(* PLC project mixture, Dassault Systèmes ControlBuild 2024x *)
(* stored: creationDateTime 2023-10-03T11:13:39-01:00 *)

FUNCTION_BLOCK faults
  VAR_INPUT
    generalFault1 : BOOL := false;
    generalFault2 : BOOL := false;
    generalFault3 : BOOL := false;
  END_VAR
  VAR_OUTPUT
    fault : BOOL := false;
  END_VAR

(* LD diagram, written out as Structured Text *)
1:
fault := generalFault3 OR generalFault1 OR generalFault2;
END_FUNCTION_BLOCK

PROGRAM batch.mixture
  VAR_INPUT
    cycleInProgress : BOOL := false;
    kneadingRequest : BOOL := false;
    acknowledgePB : BOOL := false;
  END_VAR
  VAR_INPUT
    autoMode : BOOL := false;
    manualMode : BOOL := false;
  END_VAR
  VAR_INPUT
    syrupExtraction : REAL := 0.0;
    flourExtraction : REAL := 0.0;
  END_VAR
  VAR_OUTPUT
    kneadingOK : BOOL := false;
    fault : BOOL := false;
  END_VAR

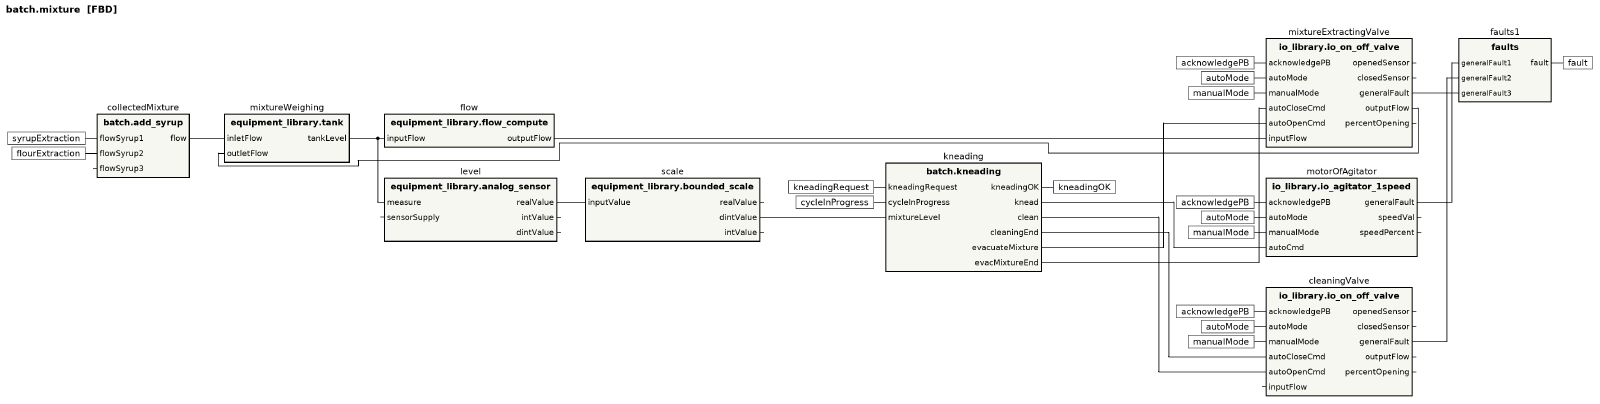
(* FBD diagram, written out as Structured Text *)
collectedMixture(flowSyrup1 := syrupExtraction, flowSyrup2 := flourExtraction);
flow(inputFlow := mixtureWeighing.tankLevel);
mixtureExtractingValve(acknowledgePB := acknowledgePB, autoMode := autoMode, manualMode := manualMode, autoCloseCmd := kneading.evacMixtureEnd, autoOpenCmd := kneading.evacuateMixture, inputFlow := flow.outputFlow);
mixtureWeighing(inletFlow := collectedMixture.flow, outletFlow := mixtureExtractingValve.outputFlow);
level(measure := mixtureWeighing.tankLevel);
scale(inputValue := level.realValue);
kneading(kneadingRequest := kneadingRequest, cycleInProgress := cycleInProgress, mixtureLevel := scale.dintValue);
kneadingOK := kneading.kneadingOK;
motorOfAgitator(acknowledgePB := acknowledgePB, autoMode := autoMode, manualMode := manualMode, autoCmd := kneading.knead);
cleaningValve(acknowledgePB := acknowledgePB, autoMode := autoMode, manualMode := manualMode, autoCloseCmd := kneading.cleaningEnd, autoOpenCmd := kneading.clean);
faults1(generalFault1 := motorOfAgitator.generalFault, generalFault2 := cleaningValve.generalFault, generalFault3 := mixtureExtractingValve.generalFault);
fault := faults1.fault;
END_PROGRAM
